// TIA Portal V21 export
DATA_BLOCK "DB625"   // DB625
TITLE = REPORT PROCESS VALUE
{ S7_Optimized_Access := 'FALSE' }
// stored: AutoNumber false
   VAR RETAIN
      RepetitionPrint : Array[0..3] of Int;
      FillingPrint : Array[0..3] of "FillingPrint";
      MixingTime { S7_SetPoint := 'True'} : Array[0..3] of "MixingPrint";
      Pulsingtime { S7_SetPoint := 'True'} : Array[0..3] of "PulsingPrint";
      spare { S7_SetPoint := 'True'} : Bool;
      RecirculationPrint { S7_SetPoint := 'True'} : Array[0..3] of "RecirculationPrint";
      DrainPrint { S7_SetPoint := 'True'} : Array[0..3] of "DrainPrint";
      ConductivityStatus { S7_SetPoint := 'True'} : Array[0..3] of Bool;
   END_VAR
BEGIN
END_DATA_BLOCK
